// TIA Portal V21 export
DATA_BLOCK "AzionamentoFesto"   // DB14
{ S7_Optimized_Access := 'TRUE' }
// stored: MemoryReserve 100
   VAR RETAIN
      AF : Array[0..1] of "Std_Azionamentofesto";
   END_VAR
BEGIN
   // AF[0] : Non usare
   // AF[1] : AltezzaStampo
   AF[0].Input.ModePos := 0;
   AF[1].Input.ModePos := 7;
   AF[0].Input.EnableAxis := FALSE;
   AF[1].Input.EnableAxis := TRUE;
   AF[0..1].Input.CancelTraversing := TRUE;
   AF[0..1].Input.IntermediateStop := TRUE;
   AF[0..1].Input.Positive := FALSE;
   AF[0..1].Input.Negative := FALSE;
   AF[0..1].Input.Jog1 := FALSE;
   AF[0..1].Input.Jog2 := FALSE;
   AF[0..1].Input.AckError := FALSE;
   AF[0..1].Input.ExecuteMode := FALSE;
   AF[0..1].Input.ReleaseBrake := FALSE;
   AF[0..1].Input.TravelToFixStop := FALSE;
   AF[0].Input.Position := 0;
   AF[1].Input.Position := 120000;
   AF[0..1].Input.Velocity := 0;
   AF[0..1].Input.OverV := 100;
   AF[0..1].Input.OverAcc := 100;
   AF[0..1].Input.OverDec := 100;
   AF[0..1].Input.ConfigEPos := 16#0000_000F;
   AF[0].Input.BaseSpeedValue := 0.0;
   AF[1].Input.BaseSpeedValue := 0.042;
   AF[0].Input.HardwareId := 0;
   AF[1].Input.HardwareId := 285;
   AF[0..1].Output.AxisEnabled := FALSE;
   AF[0..1].Output.AxisPosOk := FALSE;
   AF[0..1].Output.AxisSpFixed := FALSE;
   AF[0..1].Output.AxisAckSetpoint := FALSE;
   AF[0..1].Output.ClampTorqueReached := FALSE;
   AF[0..1].Output.AxisRef := FALSE;
   AF[0..1].Output.AxisWarn := FALSE;
   AF[0..1].Output.AxisError := FALSE;
   AF[0..1].Output.Lockout := FALSE;
   AF[0..1].Output.ActVelocity := 0.0;
   AF[0..1].Output.ActPosition := 0;
   AF[0].Output.ActMode := 0;
   AF[1].Output.ActMode := 4;
   AF[0..1].Output.EPosZSW1 := 16#0000;
   AF[0..1].Output.EPosZSW2 := 16#0000;
   AF[0..1].Output.ActWarn := 16#0000;
   AF[0..1].Output.ActFault := 16#0000;
   AF[0..1].Output.Error := FALSE;
   AF[0..1].Output.Status := 16#0000;
   AF[0..1].Output.DiagID := 16#0000;
   AF[0..1].Dati.Ready4Motion := FALSE;
   AF[0..1].Dati.ExecuteIntern := FALSE;
   AF[0..1].Dati.StepHome := 0;
   AF[0..1].Dati.RetDPRD := 0;
   AF[0..1].Dati.RetDPWR := 0;
   AF[0..1].Dati.CycWrite.STW1.jog1 := FALSE;
   AF[0..1].Dati.CycWrite.STW1.jog2 := FALSE;
   AF[0..1].Dati.CycWrite.STW1.controlByPlc := TRUE;
   AF[0..1].Dati.CycWrite.STW1.StartHoming := FALSE;
   AF[0..1].Dati.CycWrite.STW1.ReleaseBrake := FALSE;
   AF[0..1].Dati.CycWrite.STW1.ExternalBlockChange := FALSE;
   AF[0..1].Dati.CycWrite.STW1.reserved14 := FALSE;
   AF[0..1].Dati.CycWrite.STW1.reserved15 := FALSE;
   AF[0..1].Dati.CycWrite.STW1.on := FALSE;
   AF[0..1].Dati.CycWrite.STW1.noCoastStop := TRUE;
   AF[0..1].Dati.CycWrite.STW1.noQuickStop := TRUE;
   AF[0..1].Dati.CycWrite.STW1.enableOperation := TRUE;
   AF[0..1].Dati.CycWrite.STW1.cancelTraversing := FALSE;
   AF[0..1].Dati.CycWrite.STW1.intermediateStop := FALSE;
   AF[0..1].Dati.CycWrite.STW1.activateTraversing := FALSE;
   AF[0..1].Dati.CycWrite.STW1.acknowledgeFault := FALSE;
   AF[0..1].Dati.CycWrite.POS_STW1.MDI_MOD := FALSE;
   AF[0..1].Dati.CycWrite.POS_STW1.PosModulo := FALSE;
   AF[0..1].Dati.CycWrite.POS_STW1.NegModulo := FALSE;
   AF[0..1].Dati.CycWrite.POS_STW1.reserved11 := FALSE;
   AF[0..1].Dati.CycWrite.POS_STW1.reserved12 := FALSE;
   AF[0..1].Dati.CycWrite.POS_STW1.reserved13 := FALSE;
   AF[0..1].Dati.CycWrite.POS_STW1.SetupMode := FALSE;
   AF[0..1].Dati.CycWrite.POS_STW1.MDI_Activate := FALSE;
   AF[0..1].Dati.CycWrite.POS_STW1.travBlockBit0 := FALSE;
   AF[0..1].Dati.CycWrite.POS_STW1.travBlockBit1 := FALSE;
   AF[0..1].Dati.CycWrite.POS_STW1.travBlockBit2 := FALSE;
   AF[0..1].Dati.CycWrite.POS_STW1.travBlockBit3 := FALSE;
   AF[0..1].Dati.CycWrite.POS_STW1.travBlockBit4 := FALSE;
   AF[0..1].Dati.CycWrite.POS_STW1.travBlockBit5 := FALSE;
   AF[0..1].Dati.CycWrite.POS_STW1.travBlockBit6 := FALSE;
   AF[0..1].Dati.CycWrite.POS_STW1.reserved7 := FALSE;
   AF[0..1].Dati.CycWrite.POS_STW2.FlyingRef := FALSE;
   AF[0..1].Dati.CycWrite.POS_STW2.reserved9 := FALSE;
   AF[0..1].Dati.CycWrite.POS_STW2.SelectProbe := FALSE;
   AF[0..1].Dati.CycWrite.POS_STW2.ProbeEdgeEval := FALSE;
   AF[0..1].Dati.CycWrite.POS_STW2.reserved12 := FALSE;
   AF[0..1].Dati.CycWrite.POS_STW2.reserved13 := FALSE;
   AF[0..1].Dati.CycWrite.POS_STW2."SW-Limit" := FALSE;
   AF[0..1].Dati.CycWrite.POS_STW2."HW-Limit" := FALSE;
   AF[0..1].Dati.CycWrite.POS_STW2.Trackingmode := FALSE;
   AF[0..1].Dati.CycWrite.POS_STW2.SetReferencePoint := FALSE;
   AF[0..1].Dati.CycWrite.POS_STW2.reserved2 := FALSE;
   AF[0..1].Dati.CycWrite.POS_STW2.reserved3 := FALSE;
   AF[0..1].Dati.CycWrite.POS_STW2.reserved4 := FALSE;
   AF[0..1].Dati.CycWrite.POS_STW2.jog_inc := FALSE;
   AF[0..1].Dati.CycWrite.POS_STW2.reserved6 := FALSE;
   AF[0..1].Dati.CycWrite.POS_STW2.reserved7 := FALSE;
   AF[0..1].Dati.CycWrite.STW2.TravelToFixStop := FALSE;
   AF[0..1].Dati.CycWrite.STW2.reserved9 := FALSE;
   AF[0..1].Dati.CycWrite.STW2.reserved10 := FALSE;
   AF[0..1].Dati.CycWrite.STW2.reserved11 := FALSE;
   AF[0..1].Dati.CycWrite.STW2.signOfLifeBit0 := FALSE;
   AF[0..1].Dati.CycWrite.STW2.signOfLifeBit1 := FALSE;
   AF[0..1].Dati.CycWrite.STW2.signOfLifeBit2 := FALSE;
   AF[0..1].Dati.CycWrite.STW2.signOfLifeBit3 := FALSE;
   AF[0..1].Dati.CycWrite.STW2.reserved0 := FALSE;
   AF[0..1].Dati.CycWrite.STW2.reserved1 := FALSE;
   AF[0..1].Dati.CycWrite.STW2.reserved2 := FALSE;
   AF[0..1].Dati.CycWrite.STW2.reserved3 := FALSE;
   AF[0..1].Dati.CycWrite.STW2.reserved4 := FALSE;
   AF[0..1].Dati.CycWrite.STW2.reserved5 := FALSE;
   AF[0..1].Dati.CycWrite.STW2.reserved6 := FALSE;
   AF[0..1].Dati.CycWrite.STW2.reserved7 := FALSE;
   AF[0..1].Dati.CycWrite.Override := 16#0000;
   AF[0..1].Dati.CycWrite.MDI_TARPOS := 0;
   AF[0..1].Dati.CycWrite.MDI_VELOCITY := 0;
   AF[0..1].Dati.CycWrite.MDI_ACC := 0;
   AF[0..1].Dati.CycWrite.MDI_DEC := 0;
   AF[0..1].Dati.CycWrite.reserved11 := 16#0000;
   AF[0..1].Dati.CycRead.ZSW1.followingErrorInTolerance := FALSE;
   AF[0..1].Dati.CycRead.ZSW1.controlRequest := FALSE;
   AF[0..1].Dati.CycRead.ZSW1.targetPosReached := FALSE;
   AF[0..1].Dati.CycRead.ZSW1.homePosSet := FALSE;
   AF[0..1].Dati.CycRead.ZSW1.acknowledgeTraversingBlockActivated := FALSE;
   AF[0..1].Dati.CycRead.ZSW1.driveStopped := FALSE;
   AF[0..1].Dati.CycRead.ZSW1.axisAccelerates := FALSE;
   AF[0..1].Dati.CycRead.ZSW1.axisDecelerates := FALSE;
   AF[0..1].Dati.CycRead.ZSW1.readyForSwitchOn := FALSE;
   AF[0..1].Dati.CycRead.ZSW1.ready := FALSE;
   AF[0..1].Dati.CycRead.ZSW1.operationEnabled := FALSE;
   AF[0..1].Dati.CycRead.ZSW1.faultPresent := FALSE;
   AF[0..1].Dati.CycRead.ZSW1.noCoastingActive := FALSE;
   AF[0..1].Dati.CycRead.ZSW1.noQuickStopActive := FALSE;
   AF[0..1].Dati.CycRead.ZSW1.switchingOnInhibitedActive := FALSE;
   AF[0..1].Dati.CycRead.ZSW1.warningActive := FALSE;
   AF[0..1].Dati.CycRead.POS_ZSW1 := 16#0000;
   AF[0..1].Dati.CycRead.POS_ZSW2 := 16#0000;
   AF[0..1].Dati.CycRead.ZSW2.deviceSpecificBit8 := FALSE;
   AF[0..1].Dati.CycRead.ZSW2.deviceSpecificBit9 := FALSE;
   AF[0..1].Dati.CycRead.ZSW2.deviceSpecificBit10 := FALSE;
   AF[0..1].Dati.CycRead.ZSW2.deviceSpecificBit11 := FALSE;
   AF[0..1].Dati.CycRead.ZSW2.doSignOfLifeBit0 := FALSE;
   AF[0..1].Dati.CycRead.ZSW2.doSignOfLifeBit1 := FALSE;
   AF[0..1].Dati.CycRead.ZSW2.doSignOfLifeBit2 := FALSE;
   AF[0..1].Dati.CycRead.ZSW2.doSignOfLifeBit3 := FALSE;
   AF[0..1].Dati.CycRead.ZSW2.deviceSpecificBit0 := FALSE;
   AF[0..1].Dati.CycRead.ZSW2.deviceSpecificBit1 := FALSE;
   AF[0..1].Dati.CycRead.ZSW2.deviceSpecificBit2 := FALSE;
   AF[0..1].Dati.CycRead.ZSW2.deviceSpecificBit3 := FALSE;
   AF[0..1].Dati.CycRead.ZSW2.deviceSpecificBit4 := FALSE;
   AF[0..1].Dati.CycRead.ZSW2.deviceSpecificBit5 := FALSE;
   AF[0..1].Dati.CycRead.ZSW2.deviceSpecificBit6 := FALSE;
   AF[0..1].Dati.CycRead.ZSW2.deviceSpecificBit7 := FALSE;
   AF[0..1].Dati.CycRead.MELDW := 16#0000;
   AF[0..1].Dati.CycRead.XIST_A := 0;
   AF[0..1].Dati.CycRead.NIST_B := 0;
   AF[0..1].Dati.CycRead.Fault_Code := 16#0000;
   AF[0..1].Dati.CycRead.Warn_Code := 16#0000;
   AF[0..1].Dati.CycRead.Reserved := 16#0000;
   AF[0..1].Dati.ExecAux := FALSE;
   AF[0..1].Dati.ExecR_Trig := FALSE;
   AF[0..1].Dati.Jog1PAux := FALSE;
   AF[0..1].Dati.Jog1PR_trig := FALSE;
   AF[0..1].Dati.Jog2PAux := FALSE;
   AF[0..1].Dati.Jog2PR_trig := FALSE;
   AF[0..1].Dati.Jog1PMode8Aux := FALSE;
   AF[0..1].Dati.Jog1PMode8R_trig := FALSE;
   AF[0..1].Dati.Jog2PMode8Aux := FALSE;
   AF[0..1].Dati.Jog2PMode8R_trig := FALSE;
   AF[0..1].Dati.Status := 16#0000;
   AF[0..1].Dati.statStartCounter := 0;
   AF[0..1].Dati.ActMode := 0;
   AF[0..1].Dati.MaxCounterRetries := 0;
   AF[0..1].Dati.GestioneExecute.OldPosition := 0;
   AF[0..1].Dati.GestioneExecute.OldStatoMotore := 0;
   AF[0..1].Dati.GestioneExecute.OldAxisEnable := FALSE;
   AF[0..1].Dati.GestioneExecute.OldModePos := 0;
   AF[0..1].Dati.GestioneExecute.OldResetState := FALSE;
   AF[0..1].Dati.GestioneExecute.Richiesto := FALSE;
   AF[0..1].Dati.GestioneExecute.Attesa := 0;
   AF[0..1].Dati.GestioneExecute.Durata := 0;
END_DATA_BLOCK
